// TIA Portal V19 export
ORGANIZATION_BLOCK "Main"   // OB1, LAD, ProgramCycle
TITLE = "Main Program Sweep (Cycle)"
{ S7_Optimized_Access := 'TRUE' }
// stored: SetENOAutomatically false
   VAR_INPUT
      Initial_Call : Bool;   // Initial call of this OB
      Remanence : Bool;   // =True, if remanent data are available
   END_VAR
   VAR_TEMP   // added for the SCL form of the ladder/FBD networks
      _w1 : Bool;
      _w2 : Bool;
      _w3 : Bool;
      _w4 : Bool;
      _w5 : Bool;
      _w6 : Bool;
      _w7 : Bool;
      _w8 : Bool;
   END_VAR
BEGIN

REGION Network 1: MAIN BLOCK CALLING
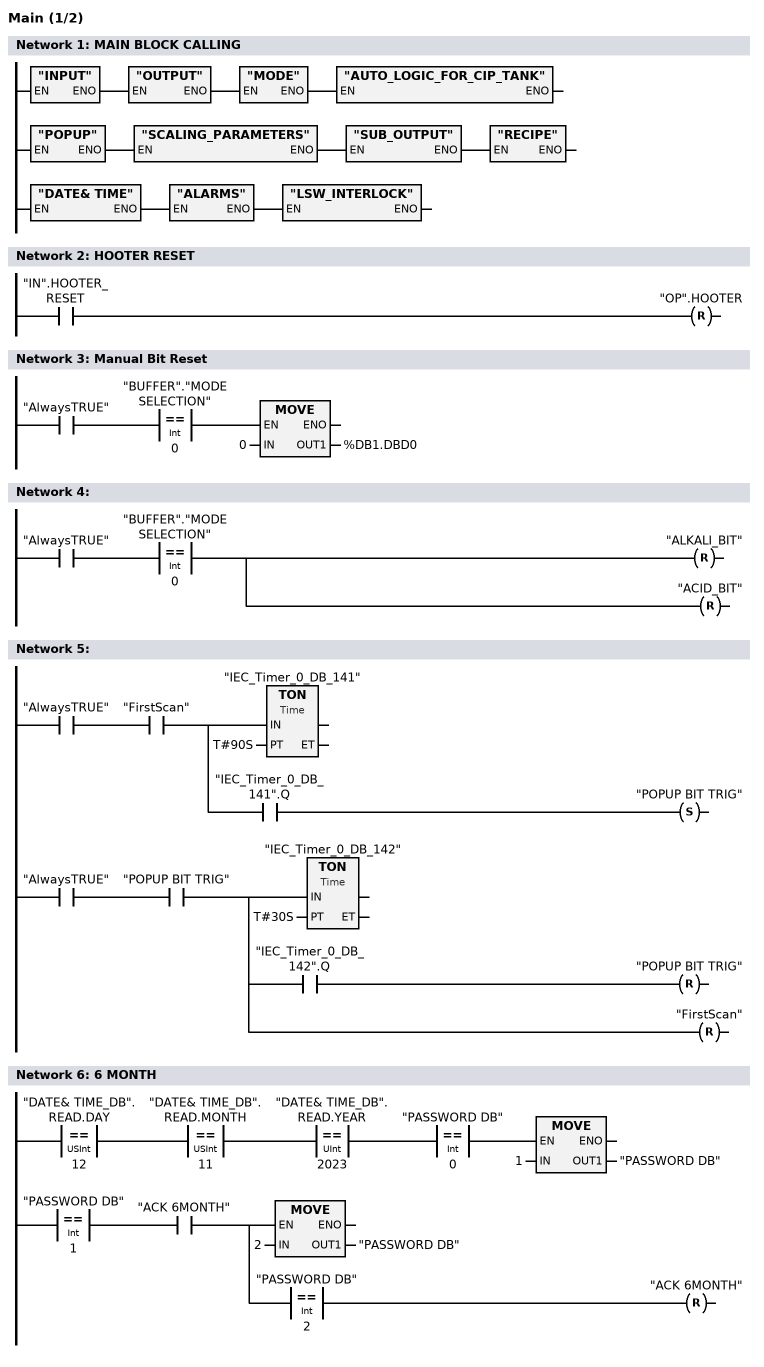
   RUNG wire#powerrail
      "INPUT"()
      "OUTPUT"()
      "MODE"()
      "AUTO_LOGIC_FOR_CIP_TANK"()
   END_RUNG
   RUNG wire#powerrail
      "POPUP"()
      "SCALING_PARAMETERS"()
      "SUB_OUTPUT"()
      "RECIPE"()
   END_RUNG
   RUNG wire#powerrail
      "DATE& TIME"()
      "ALARMS"()
      "LSW_INTERLOCK"()
   END_RUNG
   // the same network as SCL:
   "INPUT"(ENO => #_w1);
   "OUTPUT"(EN := #_w1, ENO => #_w2);
   "MODE"(EN := #_w2, ENO => #_w3);
   IF #_w3 THEN "AUTO_LOGIC_FOR_CIP_TANK"(); END_IF;
   "POPUP"(ENO => #_w4);
   "SCALING_PARAMETERS"(EN := #_w4, ENO => #_w5);
   "SUB_OUTPUT"(EN := #_w5, ENO => #_w6);
   IF #_w6 THEN "RECIPE"(); END_IF;
   "DATE& TIME"(ENO => #_w7);
   "ALARMS"(EN := #_w7, ENO => #_w8);
   IF #_w8 THEN "LSW_INTERLOCK"(); END_IF;
END_REGION

REGION Network 2: HOOTER RESET
   RUNG wire#powerrail
      Contact( "IN".HOOTER_RESET )
      R_Coil( "OP".HOOTER )
   END_RUNG
   // the same network as SCL:
   IF "IN".HOOTER_RESET THEN "OP".HOOTER := FALSE; END_IF;
END_REGION

REGION Network 3: Manual Bit Reset
   RUNG wire#powerrail
      Contact( "AlwaysTRUE" )
      { S7_Templates := "SrcType := Int" } EQ_Contact(in1 := "BUFFER"."MODE SELECTION", in2 := 0)
      Move(in := 0, out1 => %DB1.DBD0)
   END_RUNG
   // the same network as SCL:
   IF "AlwaysTRUE" AND ("BUFFER"."MODE SELECTION" = 0) THEN %DB1.DBD0 := 0; END_IF;
END_REGION

REGION Network 4
   RUNG wire#powerrail
      Contact( "AlwaysTRUE" )
      { S7_Templates := "SrcType := Int" } EQ_Contact(in1 := "BUFFER"."MODE SELECTION", in2 := 0)
      wire#w1
      R_Coil( "ALKALI_BIT" )
   END_RUNG
   RUNG wire#w1
      R_Coil( "ACID_BIT" )
   END_RUNG
   // the same network as SCL:
   IF "AlwaysTRUE" AND ("BUFFER"."MODE SELECTION" = 0) THEN
       "ALKALI_BIT" := FALSE;
       "ACID_BIT" := FALSE;
   END_IF;
END_REGION

REGION Network 5
   RUNG wire#powerrail
      Contact( "AlwaysTRUE" )
      Contact( "FirstScan" )
      wire#w1
      { S7_Templates := "time_type := Time" } "IEC_Timer_0_DB_141".TON(pt := T#90S, et =>)
   END_RUNG
   RUNG wire#w1
      Contact( "IEC_Timer_0_DB_141".Q )
      S_Coil( "POPUP BIT TRIG" )
   END_RUNG
   RUNG wire#powerrail
      Contact( "AlwaysTRUE" )
      Contact( "POPUP BIT TRIG" )
      wire#w2
      { S7_Templates := "time_type := Time" } "IEC_Timer_0_DB_142".TON(pt := T#30S, et =>)
   END_RUNG
   RUNG wire#w2
      Contact( "IEC_Timer_0_DB_142".Q )
      R_Coil( "POPUP BIT TRIG" )
   END_RUNG
   RUNG wire#w2
      R_Coil( "FirstScan" )
   END_RUNG
   // the same network as SCL:
   #_w1 := "AlwaysTRUE" AND "FirstScan";
   "IEC_Timer_0_DB_141".TON(IN := #_w1, PT := T#90S);
   IF #_w1 AND "IEC_Timer_0_DB_141".Q THEN "POPUP BIT TRIG" := TRUE; END_IF;
   #_w2 := "AlwaysTRUE" AND "POPUP BIT TRIG";
   "IEC_Timer_0_DB_142".TON(IN := #_w2, PT := T#30S);
   IF #_w2 AND "IEC_Timer_0_DB_142".Q THEN "POPUP BIT TRIG" := FALSE; END_IF;
   IF #_w2 THEN "FirstScan" := FALSE; END_IF;
END_REGION

REGION Network 6: 6 MONTH
   RUNG wire#powerrail
      { S7_Templates := "SrcType := USInt" } EQ_Contact(in1 := "DATE& TIME_DB".READ.DAY, in2 := 12)
      { S7_Templates := "SrcType := USInt" } EQ_Contact(in1 := "DATE& TIME_DB".READ.MONTH, in2 := 11)
      { S7_Templates := "SrcType := UInt" } EQ_Contact(in1 := "DATE& TIME_DB".READ.YEAR, in2 := 2023)
      { S7_Templates := "SrcType := Int" } EQ_Contact(in1 := "PASSWORD DB", in2 := 0)
      Move(in := 1, out1 => "PASSWORD DB")
   END_RUNG
   RUNG wire#powerrail
      { S7_Templates := "SrcType := Int" } EQ_Contact(in1 := "PASSWORD DB", in2 := 1)
      Contact( "ACK 6MONTH" )
      wire#w1
      Move(in := 2, out1 => "PASSWORD DB")
   END_RUNG
   RUNG wire#w1
      { S7_Templates := "SrcType := Int" } EQ_Contact(in1 := "PASSWORD DB", in2 := 2)
      R_Coil( "ACK 6MONTH" )
   END_RUNG
   // the same network as SCL:
   IF ("DATE& TIME_DB".READ.DAY = 12) AND ("DATE& TIME_DB".READ.MONTH = 11) AND ("DATE& TIME_DB".READ.YEAR = 2023) AND ("PASSWORD DB" = 0) THEN
       "PASSWORD DB" := 1;
   END_IF;
   #_w1 := ("PASSWORD DB" = 1) AND "ACK 6MONTH";
   IF #_w1 THEN "PASSWORD DB" := 2; END_IF;
   IF #_w1 AND ("PASSWORD DB" = 2) THEN "ACK 6MONTH" := FALSE; END_IF;
END_REGION

REGION Network 7: 8 MONTH
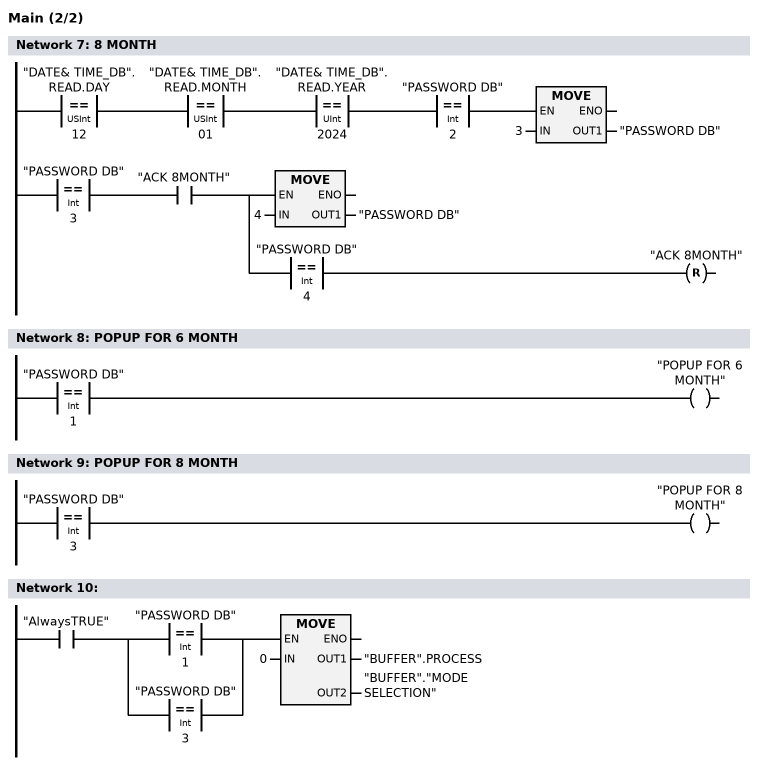
   RUNG wire#powerrail
      { S7_Templates := "SrcType := USInt" } EQ_Contact(in1 := "DATE& TIME_DB".READ.DAY, in2 := 12)
      { S7_Templates := "SrcType := USInt" } EQ_Contact(in1 := "DATE& TIME_DB".READ.MONTH, in2 := 01)
      { S7_Templates := "SrcType := UInt" } EQ_Contact(in1 := "DATE& TIME_DB".READ.YEAR, in2 := 2024)
      { S7_Templates := "SrcType := Int" } EQ_Contact(in1 := "PASSWORD DB", in2 := 2)
      Move(in := 3, out1 => "PASSWORD DB")
   END_RUNG
   RUNG wire#powerrail
      { S7_Templates := "SrcType := Int" } EQ_Contact(in1 := "PASSWORD DB", in2 := 3)
      Contact( "ACK 8MONTH" )
      wire#w1
      Move(in := 4, out1 => "PASSWORD DB")
   END_RUNG
   RUNG wire#w1
      { S7_Templates := "SrcType := Int" } EQ_Contact(in1 := "PASSWORD DB", in2 := 4)
      R_Coil( "ACK 8MONTH" )
   END_RUNG
   // the same network as SCL:
   IF ("DATE& TIME_DB".READ.DAY = 12) AND ("DATE& TIME_DB".READ.MONTH = 01) AND ("DATE& TIME_DB".READ.YEAR = 2024) AND ("PASSWORD DB" = 2) THEN
       "PASSWORD DB" := 3;
   END_IF;
   #_w1 := ("PASSWORD DB" = 3) AND "ACK 8MONTH";
   IF #_w1 THEN "PASSWORD DB" := 4; END_IF;
   IF #_w1 AND ("PASSWORD DB" = 4) THEN "ACK 8MONTH" := FALSE; END_IF;
END_REGION

REGION Network 8: POPUP FOR 6 MONTH
   RUNG wire#powerrail
      { S7_Templates := "SrcType := Int" } EQ_Contact(in1 := "PASSWORD DB", in2 := 1)
      Coil( "POPUP FOR 6 MONTH" )
   END_RUNG
   // the same network as SCL:
   "POPUP FOR 6 MONTH" := "PASSWORD DB" = 1;
END_REGION

REGION Network 9: POPUP FOR 8 MONTH
   RUNG wire#powerrail
      { S7_Templates := "SrcType := Int" } EQ_Contact(in1 := "PASSWORD DB", in2 := 3)
      Coil( "POPUP FOR 8 MONTH" )
   END_RUNG
   // the same network as SCL:
   "POPUP FOR 8 MONTH" := "PASSWORD DB" = 3;
END_REGION

REGION Network 10
   RUNG wire#powerrail
      Contact( "AlwaysTRUE" )
      wire#w1
      { S7_Templates := "SrcType := Int" } EQ_Contact(in1 := "PASSWORD DB", in2 := 1)
      wire#w2
      Move(in := 0, out1 => "BUFFER".PROCESS, out2 => "BUFFER"."MODE SELECTION")
   END_RUNG
   RUNG wire#w1
      { S7_Templates := "SrcType := Int" } EQ_Contact(in1 := "PASSWORD DB", in2 := 3)
   END_RUNG wire#w2
   // the same network as SCL:
   IF "AlwaysTRUE" AND (("PASSWORD DB" = 1) OR ("PASSWORD DB" = 3)) THEN
       "BUFFER".PROCESS := 0;
       "BUFFER"."MODE SELECTION" := 0;
   END_IF;
END_REGION
END_ORGANIZATION_BLOCK
